// TIA Portal V18 export
FUNCTION "mot_set_speed_by_target_multiturn_util1_2" : Void   // FC24, FBD
{ S7_Optimized_Access := 'TRUE' }
VERSION : 0.1
// stored: AutoNumber true, IsIECCheckEnabled false, SetENOAutomatically false, UDAEnableTagReadback false
   VAR_INPUT
      distance0 : Real;
      distance1Plus : Real;
      distance2minus : Real;
   END_VAR
   VAR_OUTPUT
      closest_0 : Bool;
      closest_1PlusTurn : Bool;
      closest_2MinusTurn : Bool;
   END_VAR
BEGIN

REGION Network 1 (SCL)
   #closest_0 := #closest_1PlusTurn := #closest_2MinusTurn := false;

   IF #distance0 <= #distance1Plus AND #distance0 <= #distance2minus THEN
       #closest_0 := true;
   ELSIF #distance1Plus <= #distance0 AND #distance1Plus <= #distance2minus THEN
       #closest_1PlusTurn := true;
   ELSE
       #closest_2MinusTurn := true;
   END_IF;
END_REGION
END_FUNCTION
